TEXTLIST TextList_STATE_Mode_Marche
  0 = '0 - PLC Off' | FR: "0 - Automate à l'arrêt" | EN: '0 - PLC Off'
  1 = '1 - PLC Starting' | FR: '1 - Démarrage automate' | EN: '1 - PLC starting'
  2 = '2 - Waiting for\nmachine supply' | FR: '2 - Attente\nalimentation machine' | EN: '2 - Waiting for machine supply'
  3 = '3 - Machine stopped' | FR: "3 - Machine à l'arrêt" | EN: '3 - Machine stopped'
  4 = '4 - Waiting for operating\nmode selection...' | FR: '4 - Attente sélection\nmode de marche...' | EN: '4 - Wait for operating mode selection...'
  5 = '5 - Machine initialization...' | FR: '5 - Initialisation machine' | EN: '5 - Machine initialization'
  6 = '6 - Automatic mode' | FR: '6 - Mode automatique' | EN: '6 - Automatic mode'
  7 = '7 - Production preparation' | FR: '7 - Préparation production' | EN: '7 - Production preparation'
  8 = '8 - Production' | FR: '8 - Production en cours...' | EN: '8 - Production in progress...'
  9 = '9 - Production stopped' | FR: '9 - Production stoppée' | EN: '9 - Production stopped'
  10 = '10 - Manual mode' | FR: '10 - Mode manuel' | EN: '10 - Manual mode'
  11 = '11 - Fin de production' | FR: '11 - Fin de production' | EN: '11 - End of production'
  12 = '12 - Interruption de production' | FR: '12 - Interruption de production' | EN: '12 - Production interruption'
  13 = '13 - En attente de reprise' | FR: '13 - En attente de reprise' | EN: '13 - Waiting for resume'
  20 = '20 - Lancement Eco' | FR: '20 - Lancement Eco Mode' | EN: '20 - Eco Mode starting'
  21 = '21 - Eco Mode' | FR: '21 - Eco Mode' | EN: '21 - Eco Mode'
  22 = '22 - Lancement procédé\neco-veille profond' | FR: '22 - Lancement procédé\neco-veille profond' | EN: '22 - Deep eco-sleep process starting'
  23 = '23 - Lancement procédé\neco-veille profond' | FR: '23 - Lancement procédé\neco-veille profond' | EN: '23 - Deep eco-sleep process starting'
  24 = '24 - Procédé eco-veille\nprofond en cours' | FR: '24 - Procédé eco-veille\nprofond en cours' | EN: '24 - Deep eco-sleep process running'
  25 = '25 - Arrêt procédé\neco-veille profond' | FR: '25 - Arrêt procédé\neco-veille profond' | EN: '25 - Deep eco-sleep process end'
  26 = '26 - Procédé eco-veille\nprofond en défaut' | FR: '26 - Procédé eco-veille\nprofond en défaut' | EN: '26 - Deep eco-sleep process in fault'
  27 = '27 - Attente sortie de veille\nappareils' | FR: '27 - Attente sortie de veille\nappareils' | EN: '27 - Waiting for devices wakes up'
   = ''
END_TEXTLIST

(* stored: Version 1.1.0.1, ProductVersion 3.1.4024.12
   TextList TextList_STATE_Mode_Marche: Id {093db9f2-2791-4b21-a7cb-f7e3999665df} *)
